TYPE "PartNumber_ShW"
VERSION : 0.1
   STRUCT
      material_id : String[28];
      lot_code : String[18];
      Quantity : Int;
      ScanOK : Bool;
   END_STRUCT;

END_TYPE

